FUNCTION ConvertMilliSecTimeData : TIME
VAR_INPUT
	DataInput	: UINT;
END_VAR
VAR
END_VAR

ConvertMilliSecTimeData:=LINT_TO_TIME(UINT_TO_LINT(DataInput));

END_FUNCTION

(* stored: Version 1.1.0.1, ProductVersion 3.1.4024.12
   POU ConvertMilliSecTimeData: Id {ef477df3-7d1c-4c33-9db5-386773a09fa8}, SpecialFunc None *)
